FUNCTION_BLOCK FB_ltBar
VAR
	bGreenLight 	AT %Q* : BOOL;
	bRedLight 		AT %Q* : BOOL;
	bYellowLight 	AT %Q* : BOOL;
END_VAR

METHOD greenOn : BOOL
VAR_INPUT
END_VAR
bGreenLight 	:= TRUE;
bRedLight 		:= FALSE;
bYellowLight 	:= FALSE;
END_METHOD

METHOD redOn : BOOL
VAR_INPUT
END_VAR
bGreenLight 	:= FALSE;
bRedLight 		:= TRUE;
bYellowLight 	:= FALSE;
END_METHOD

METHOD yellowOn : BOOL
VAR_INPUT
END_VAR
bGreenLight 	:= FALSE;
bRedLight 		:= FALSE;
bYellowLight 	:= TRUE;
END_METHOD

END_FUNCTION_BLOCK

(* stored: Version 1.1.0.1, ProductVersion 3.1.4024.13
   POU FB_ltBar: Id {5417c8d7-1356-49ab-967c-d3f0ac445e80}, SpecialFunc None
   Method greenOn: Id {a9b8a284-2195-4e8e-b537-2f4fa026cdad}
   Method redOn: Id {94556ece-180a-4955-be62-60beca4247d4}
   Method yellowOn: Id {dc4fc304-5289-40ac-9e6d-0730f3de449e} *)
